PROGRAM CommWithCamera
VAR
END_VAR

END_PROGRAM

(* stored: Version 1.1.0.1, ProductVersion 3.1.4024.9
   POU CommWithCamera: Id {19c51c70-23e6-48e7-b9f9-e1f96618f2f6}, SpecialFunc None *)
